FUNCTION_BLOCK AS_TO_AS2 (* Composite FB for convert unidirectional AS to bidirectional AS2 *)
  (* Standard: 61499-2; Function: AS_IN publishes its value onto the outgoing (EO1) side of AS2_BIDIR. Whatever AS2_BIDIR receives on its incoming (EI1) side is forwarded out again as a plain unidirectional signal via AS_OUT.; Description: Copyright (c) 2026 HR Agrartechnik GmbH This program and the accompanying materials are made available under the terms of the Eclipse Public License 2.0 which is available at https://www.eclipse.org/legal/epl-2.0/ SPDX-License-Identifier: EPL-2.0 *)
  (* Version 1.0, 2026-09-12, Franz Höpfinger, HR Agrartechnik GmbH, Initial Version - Konvertierungsfamilie vervollstaendigt (analog zu AR2/AB2/AE2). *)
  PACKAGE adapter::conversion::bidirectional;
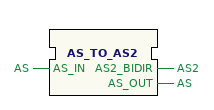
  SOCKETS
    AS_IN : adapter::types::unidirectional::AS; (* Adapter Input: unidirectional source *)
  END_SOCKETS
  PLUGS
    AS2_BIDIR : adapter::types::bidirectional::AS2; (* Adapter Output: bidirectional tap, outgoing side driven by AS_IN, incoming side forwarded to AS_OUT *)
    AS_OUT : adapter::types::unidirectional::AS; (* Adapter Output: mirrors AS2_BIDIR's incoming (request) side *)
  END_PLUGS
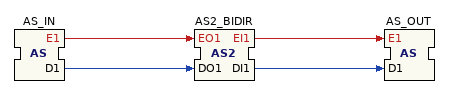
  EVENT_CONNECTIONS
    AS_IN.E1 TO AS2_BIDIR.EO1;
    AS2_BIDIR.EI1 TO AS_OUT.E1;
  END_CONNECTIONS
  DATA_CONNECTIONS
    AS_IN.D1 TO AS2_BIDIR.DO1;
    AS2_BIDIR.DI1 TO AS_OUT.D1;
  END_CONNECTIONS
END_FUNCTION_BLOCK
